// TIA Portal project "HMI" (V16)

(* hardware
DEVICE "Panel"  TP700 Comfort
   slot 0: "Panel"  TP700 Comfort  6AV2 124-0GC01-0AX0  15.1.0.0
   slot 1: "HMI_RT_1"  TP700 Comfort  6AV2 124-0GC01-0AX0  15.1.0.0
   slot 5: "Panel.IE_CP_1"  PROFINET Interface  15.0.1.0
      slot 1: "PROFINET Interface_1"  PROFINET Interface
         slot 1: "Port_1"  Port
         slot 2: "Port_2"  Port
   slot 7: "Panel.MPI/DP_CP_1"  MPI/DP Interface  15.0.1.0
DEVICE "PC station"  SIMATIC PC station
   slot 0: "PC station"  Rail  SIMATIC PC-Station  V1.0
      slot 125: "Stationmanager"  Station_Manager  V6.0.4
   slot 1: "IE general_1"  IE General  IE_CP  V8.2.0
   slot 2: "HMI_RT_2"  WinCC RT Advanced  6AV2 104-0xxxx-xxxx  16.0.0.0
      slot 33792: "Computer interface"  Host interface
DEVICE "S71500/ET200MP station_1"  S7-1500 station
   slot 0: "Rail_0"  Rack  6ES7 590-1***0-0AA0
   slot 1: "PLC_1"  CPU 1511-1 PN  6ES7 511-1AK02-0AB0  V2.8
      slot 3: "CPU display_1"  6ES7591-1AA00-0AA0
      slot 32768: "PROFINET interface_1"  X1
         slot 32769: "Port_1"  X1 P1
         slot 32770: "Port_2"  X1 P2
      slot 34817: "Virtual CP interface port_1"  Virtual CP interface port  Virtual CP interface port
*)

// ===== PLC "PLC_1"  CPU 1511-1 PN =====

VAR_GLOBAL   // PLC tag table "Default tag table"
   "HMI_Button" AT %I0.0 : Bool;
END_VAR

ORGANIZATION_BLOCK "Main"   // OB1, LAD, ProgramCycle
TITLE = "Main Program Sweep (Cycle)"
{ S7_Optimized_Access := 'TRUE' }
VERSION : 0.1
   VAR_INPUT
      Initial_Call : Bool;   // Initial call of this OB
      Remanence : Bool;   // =True, if remanent data are available
   END_VAR
BEGIN
END_ORGANIZATION_BLOCK

(* ===== HMI "HMI_RT_1" =====
system functions are stored by id; their names below are inferred from use
connection "HMI_Connection_1": ETHERNET, S7_1500_OMS

HMI tags "Default tag table"
   "HMI_Button" : Bool = PLC HMI_Button AT %I0.0, 1 s

HMI tags "Demo Tags"
   "Bit_1" : Bool, internal
   "Bit_2" : Bool, internal
   "Word_1" : Int, internal
   "Word_2" : Int, internal
   "AlarmTrigerWord" : UInt, internal
   "CurentUserName:" : WString[254], internal
   "CurentGroupNo" : Int, internal

discrete alarms
   1: 'Alarm1', class Errors, trigger "AlarmTrigerWord" bit 0
   2: 'Alarm2', class Errors, trigger "AlarmTrigerWord" bit 1
   3: 'Warnings', class Warnings, trigger "AlarmTrigerWord" bit 2
   4: 'Warnings', class Warnings, trigger "AlarmTrigerWord" bit 3

text list "OFF_ON_List": 0 'OFF'; 1 'ON'

recipe "Recipe_1": Recipe_element_1 <- "Word_1", Recipe_element_2 <- "Word_2"

SlideinScreen "GraphX_Slidein_Left" 340x480
   TextField "Text field_1" at 5,3 size 290x23; Text 'Slide in from left screen'
   Button "Button_1" at 5,441 size 258x32; TextOff 'Close'
      on Press: function_cf6f4242("GraphX_Slidein_Left", 0)

Template "ScrNav" 800x435
   Button "Template_Button_1" at 8,395 size 192x32; TextOff 'Home'
      on Click: ActivateScreen("Home", 0)
   Button "Template_Button_2" at 206,394 size 192x32; TextOff 'Toolbox'
      on Click: ActivateScreen("Toolbox", 0)
   Button "Template_Button_3" at 405,393 size 192x32; TextOff 'Alarms'
      on Click: ActivateScreen("Alarms", 0)
   Button "Template_Button_4" at 603,393 size 192x32; TextOff 'Trend'
      on Click: ActivateScreen("Trend", 0)
   Button "Template_Button_5" at 9,357 size 192x32; TextOff 'Recipe'
      on Click: ActivateScreen("Recipe", 0)
   Button "Template_Button_6" at 206,357 size 192x32; TextOff 'UserAdmin'
      on Click: ActivateScreen("UserAdmin", 0)

screen "Home" 800x435, template "ScrNav"
   TextField "Text field_1" at 593,19 size 171x23; Text 'Home Screen'
   Button "Button_1" at 14,10 size 227x32; TextOff 'Help Puop'
      on Click: function_efd93a16("Help Puop", 0, 0, 1, -1, 1)
   Button "Button_2" at 14,50 size 225x32; TextOff 'Show slide in left'
      on Press: function_cf6f4242("GraphX_Slidein_Left", 1)

screen "Toolbox" 800x435, template "ScrNav"
   Button "Button_1" at 34,18 size 225x113; TextOff 'Momentary'; TextList "OFF_ON_List"
      on Press: function_b14e0dd5("Bit_1", 0)
      Appearance <- "Bit_1"
      ProcessValue <- "Bit_1"
   IOField "I/O field_2" at 284,18 size 117x114; FormatPattern 1
      ProcessValue <- "Bit_1"
   TextField "Text field_1" at 593,19 size 193x23; Text 'Toolbox Screen'
   Circle "Circle_1" at 446,32 size 72x72
      Visibility <- "Bit_1"
   SymbolicIOField "Symbolic I/O field_1" at 545,55 size 170x66; TextOff '0'; TextOn '1'; TextList "OFF_ON_List"
      ProcessValue <- "Bit_1"

PopupScreen "Help Puop" 240x240
   Button "Button_1" at 3,200 size 229x32; TextOff 'Close'
      on Press: function_efd93a16("Help Puop", 0, 0, 0, -1, 1)
   TextField "Text field_2" at 8,8 size 107x23; Text 'Help popup'

screen "Alarms" 800x435, template "ScrNav"
   TextField "Text field_1" at 17,6 size 233x23; Text 'Alarm Trigher Word Bits:'
   IOField "I/O field_1" at 261,10 size 96x32; FormatPattern 1111
      ProcessValue <- "AlarmTrigerWord"
   TextField "Text field_2" at 593,19 size 174x23; Text 'Alarm Screen'
   AlarmView "Alarm view_1" at 12,46 size 756x178
   AlarmView "Alarm view_2" at 13,229 size 755x159

screen "Trend" 800x435, template "ScrNav"
   IOField "I/O field_1" at 143,20 size 96x32; FormatPattern s99999
      ProcessValue <- "Word_1"
   TextField "Text field_1" at 27,23 size 74x23; Text 'Word_1'
   TextField "Text field_2" at 301,23 size 74x23; Text 'Word_2'
   IOField "I/O field_2" at 427,23 size 96x32; FormatPattern s99999
      ProcessValue <- "Word_2"
   TextField "Text field_3" at 593,19 size 173x23; Text 'Trend Screen'
   RecipeView "Recipe view_1" at 11,46 size 780x307

screen "Recipe" 800x435, template "ScrNav"
   IOField "I/O field_1" at 143,20 size 96x32; FormatPattern s99999
      ProcessValue <- "Word_1"
   TextField "Text field_1" at 27,23 size 74x23; Text 'Word_1'
   TextField "Text field_2" at 301,23 size 74x23; Text 'Word_2'
   IOField "I/O field_2" at 427,23 size 96x32; FormatPattern s99999
      ProcessValue <- "Word_2"
   TextField "Text field_3" at 593,19 size 181x23; Text 'Recipe Screen'
   RecipeView "Recipe view_1" at 8,53 size 782x299

screen "UserAdmin" 800x435, template "ScrNav"
   IOField "I/O field_1" at 114,24 size 96x32; Authorization "Operate"; FormatPattern s99999
      ProcessValue <- "Word_1"
   TextField "Text field_1" at 27,23 size 74x23; Text 'Word_1'
   TextField "Text field_2" at 252,24 size 177x23; Text 'Curent User Name:'
   TextField "Text field_3" at 251,68 size 163x23; Text 'Curent Group No:'
   TextField "Text field_4" at 593,19 size 218x23; Text 'UserAdmin Screen'
   Button "Button_1" at 652,56 size 131x47; TextOff 'Login'
      on Press: function_a2a04561()
   Button "Button_2" at 652,117 size 131x47; TextOff 'Logoff'
      on Press: function_f23ef4c9()
   Button "Button_3" at 665,228 size 118x36; TextOff 'Clear Msgs'
   IOField "I/O field_2" at 445,64 size 96x32; FormatPattern s99999
      ProcessValue <- "CurentGroupNo"
   IOField "I/O field_3" at 445,23 size 95x32; FormatPattern ????????????????????????????????????????????????????????????????????????????????
      ProcessValue <- "CurentUserName:"
   UserView "User view_1" at 4,98 size 643x123
   AlarmView "Alarm view_2" at 3,230 size 643x159

scheduled task "ChgUserTask"
   on Action: function_f41c6f6c("CurentUserName:"); function_e1ab61de("CurentGroupNo")
*)